KUKA KRL program: friBare_RT.src, friBare_RT.dat

--- friBare_RT.src ---
&ACCESS RVP
&REL 16
&PARAM TEMPLATE = C:\KRC\Roboter\Template\vorgabe
&PARAM EDITMASK = *
DEF friBare_RT( )
;FOLD INI
  ;FOLD BASISTECH INI
    GLOBAL INTERRUPT DECL 3 WHEN $STOPMESS==TRUE DO IR_STOPM ( )
    INTERRUPT ON 3
    BAS (#INITMOV,0 )
  ;ENDFOLD (BASISTECH INI)
  ;FOLD USER INI
    ;Make your modifications here


  ;ENDFOLD (USER INI)
;ENDFOLD (INI)
for i=1 to 16
$fri_to_int[i]=0
$fri_to_rea[i]=0.0
endfor

bas(#tool,2)
halt ;input correct tool number here and restart


;move to Home-Position
;some movement is essential to release the brakes
ptp { a1 0,a2 147,a3 90,a4 -10,a5 -44,a6 0,e1 -100}
HALT

; Test open FRI with datarate 1 msec
retVal=friopen(1)
wait for ($FriState==#MON)
$fri_to_int[1]=0
$fri_to_rea[1]=0.123
$stiffness.strategy=30;
$stiffness.axismaxdeltatrq={A1 100, A2 100, A3 100, A4 100, A5 100, A6 30, E1 30}
$stiffness.commit=true;
wait for ($FriQuality==#PERFECT)
retVal=FRISTART(1.0)
wait for ($FriState==#CMD)

halt
;FOLD PTP P4 Vel=100 % PDAT4 Tool[1]:no_tool Base[0];%{PE}%R 5.6.11,%MKUKATPBASIS,%CMOVE,%VPTP,%P 1:PTP, 2:P4, 3:, 5:100, 7:PDAT4
$BWDSTART=FALSE
PDAT_ACT=PPDAT4
FDAT_ACT=FP4
BAS(#PTP_PARAMS,100)
PTP XP4
;ENDFOLD

END

--- friBare_RT.dat ---
&ACCESS RVP
&REL 16
&PARAM TEMPLATE = C:\KRC\Roboter\Template\vorgabe
&PARAM EDITMASK = *
DEFDAT  FRIBARE_RT
;FOLD EXTERNAL DECLARATIONS;%{PE}%MKUKATPBASIS,%CEXT,%VCOMMON,%P
;FOLD BASISTECH EXT;%{PE}%MKUKATPBASIS,%CEXT,%VEXT,%P
EXT  BAS (BAS_COMMAND  :IN,REAL  :IN )
DECL INT SUCCESS
;ENDFOLD (BASISTECH EXT)
;FOLD USER EXT;%{E}%MKUKATPUSER,%CEXT,%VEXT,%P
;Make here your modifications

INT i
DECL FRISTATE retVal

;ENDFOLD (USER EXT)
;ENDFOLD (EXTERNAL DECLERATIONS)
DECL BASIS_SUGG_T LAST_BASIS={POINT1[] "P4                      ",POINT2[] "P4                      ",CP_PARAMS[] "CPDAT0                  ",PTP_PARAMS[] "PDAT4                   ",CONT[] "                        ",CP_VEL[] "2.0                     ",PTP_VEL[] "100                     ",SYNC_PARAMS[] "SYNCDAT                 ",SPL_NAME[] "S0                      "}
DECL E6POS XP3={X 1521.84802,Y 119.7743,Z 350.667206,A -178.071503,B 66.9796371,C 177.632904,S 6,T 24,E1 -0.000360488892,E2 0.0,E3 0.0,E4 0.0,E5 0.0,E6 0.0}
DECL FDAT FP3={TOOL_NO 1,BASE_NO 0,IPO_FRAME #BASE,POINT2[] " ",TQ_STATE FALSE}
DECL PDAT PPDAT3={VEL 100.0,ACC 100.0,APO_DIST 100.0}
DECL E6POS XP4={X 52.5444603,Y -1344.57202,Z -94.9417267,A 51.6422501,B 37.9400902,C 134.232101,S 7,T 57,E1 -88.0715408,E2 0.0,E3 0.0,E4 0.0,E5 0.0,E6 0.0}
DECL FDAT FP4={TOOL_NO 1,BASE_NO 0,IPO_FRAME #BASE,POINT2[] " ",TQ_STATE FALSE}
DECL PDAT PPDAT4={VEL 100.0,ACC 100.0,APO_DIST 100.0}
ENDDAT
